FUNCTION_BLOCK EL1852
VAR
	_io : EL1852_Data;
	{attribute addProperty Name "WcState"}
	_wcState : WcStateInputToggle;
	{attribute addProperty Name "Info data"}
	_infoData : InfoDataBase;
END_VAR

PROPERTY IO : REFERENCE TO EL1852_Data
GET
IO REF= _io;
END_GET
END_PROPERTY

PROPERTY WcState : REFERENCE TO WcStateInputToggle
GET
WcState REF= _wcState;
END_GET
END_PROPERTY

END_FUNCTION_BLOCK

(* stored: Version 1.1.0.1, ProductVersion 3.1.4024.9
   POU EL1852: Id {bb4d4acb-152a-0c50-2320-5e1213478461}, SpecialFunc None
   Property IO: Id {32513370-056b-074a-2ae2-853942cf88e9}
   Get Get: Id {e38ab64c-f18c-0485-2c79-85e58aa83426}
   Property WcState: Id {7f3f956c-ca84-06a4-0f71-3fa3a6645423}
   Get Get: Id {c4a72177-5c08-0088-225b-3a47f6e4f5a5} *)
